PROGRAM MAIN
VAR
	fbCreateFolder : FB_CreateFolder(sNetID := '', sBasePath := 'C:\createFoldertest\');
	fbUpdateSystemTime : FB_UpdateCurrentSystemTime;
	sPathTest : T_MaxString  := 'C:\test';
	step : INT;
	TimeStruct : TIMESTRUCT;
	bInit: BOOL;
	calTimeStruct : CalculateTimeStruct;
	bTest: BOOL;
END_VAR

fbUpdateSystemTime();
IF bInit THEN
	bInit := FALSE;
	TIMESTRUCT := fbUpdateSystemTime.updatedSystemTime;
END_IF

CASE step OF
	5:
		fbCreateFolder.SetTimeStruct(TIMESTRUCT);
		fbCreateFolder.CreateYearFolder();
		IF fbCreateFolder.isCreatedYearFolder THEN
			step := 8;
		END_IF
	
	6:
		fbCreateFolder.SetTimeStruct(TIMESTRUCT);
		fbCreateFolder.CreateYearMonthDayFolder();
		IF fbCreateFolder.isCreatedYearMonthDayFolder THEN
			step := 8;
		END_IF
	
	7:
		fbCreateFolder.SetTimeStruct(TIMESTRUCT);
		fbCreateFolder.CreateYearMonthFolder();	
		IF fbCreateFolder.isCreatedYearMonthFolder THEN
			step := 8;
		END_IF

	
	8:
		TIMESTRUCT.wYear := TIMESTRUCT.wYear + 1;
		calTimeStruct(TimeStruct := TimeStruct);
		step := 5;	
END_CASE



(*------------------------------------ TEST ------------------------------------------------*)

END_PROGRAM

(* stored: Version 1.1.0.1, ProductVersion 3.1.4024.12
   POU MAIN: Id {950fdb80-d0b4-429a-ae50-eca2f5b2f0cf}, SpecialFunc None *)
